ads_router_status_record_interval_timer(IN := NOT ads_router_status_record_interval_timer.Q);
fb_get_router_status_report := fb_get_router_status.bBusy;
fb_get_router_status(
	bExecute := ads_router_status_record_interval_timer.Q
);

IF fb_get_router_status_report AND NOT fb_get_router_status.bBusy THEN
	MEMCPY(ADR(router_status_record_data), ADR(fb_get_router_status.info), SIZEOF(fb_get_router_status.info));
	IF GVL.tf6420_enable THEN
		fb_ads_router_status_recorder.write(ADR(router_status_record_data));
	END_IF
END_IF

SetDynamics := GVL.planar_movers[1].MCTOPLC.SET;
ActDynamics := GVL.planar_movers[1].MCTOPLC.ACT;

record_data_set_positions.a := SetDynamics.SetPos.a;
record_data_set_positions.b := SetDynamics.SetPos.b;
record_data_set_positions.c := SetDynamics.SetPos.c;
record_data_set_positions.x := SetDynamics.SetPos.x;
record_data_set_positions.y := SetDynamics.SetPos.y;
record_data_set_positions.z := SetDynamics.SetPos.z;

IF GVL.tf6420_enable THEN
	fb_mover_dynamics_recorder.write(ADR(record_data_set_positions));
END_IF

record_data_act_positions.a := ActDynamics.ActPos.a;
record_data_act_positions.b := ActDynamics.ActPos.b;
record_data_act_positions.c := ActDynamics.ActPos.c;
record_data_act_positions.x := ActDynamics.ActPos.x;
record_data_act_positions.y := ActDynamics.ActPos.y;
record_data_act_positions.z := ActDynamics.ActPos.z;

IF GVL.tf6420_enable THEN
	fb_mover_dynamics_recorder.write(ADR(record_data_act_positions));
END_IF

END_PROGRAM

// ---- POUs/model/IoT/FB_mqtt_publish.TcPOU
FUNCTION_BLOCK FB_mqtt_publish IMPLEMENTS  ITF_CoeSdoEventHandler
VAR_INPUT
END_VAR
VAR_OUTPUT
	fb_database_aps_diag    :ST_database_aps_diag;    // 書込みデータ設定用
END_VAR
VAR
	// published message
	fbMqttClient : FB_IotMqttClient;
	fbMessageQueue : FB_IotMqttMessageQueue;
	bSetParameter : BOOL := TRUE;
	bConnect : BOOL := TRUE;
	hrErrorOccurred : HRESULT; // contains the latest occurred error
	
	fbSerializer :FB_Serializer;
	
	sTopicPub : STRING(255) := 'devices/unit230/messages/events/';
	
	// for making publish event
	publish_cycle_timer :TON;
	datetime_string: STRING(39);
	
	publish_command: BOOL;
	_error_id :UDINT;
	
	_fbDatabaseRecorder : REFERENCE TO BufferedRecord;
	
END_VAR


// Connect MQTT broker and publish

IF bSetParameter THEN
	bSetParameter := FALSE;
	fbMqttClient.sHostName := 'IndustrialOPNFair2024-IoTHub.azure-devices.net';
	fbMqttClient.nHostPort := 8883;
	fbMqttClient.stTLS.sCA := 'c:\TwinCAT\3.1\Config\Certificates\BaltimoreCyberTrust.cer'; // CA certificate 
	fbMqttClient.sClientId := 'unit230';
	fbMqttClient.stTLS.sAzureSas := 'HostName=IndustrialOPNFair2024-IoTHub.azure-devices.net;DeviceId=unit230;SharedAccessSignature=SharedAccessSignature sr=IndustrialOPNFair2024-IoTHub.azure-devices.net%2Fdevices%2Funit230&sig=aZHGqBLbPbZ0nCj3%2BrwgAJAAhzI2BvVoTXPMA%2BaobPA%3D&se=1734308970'; // Device SAS Token
	fbMqttClient.stTLS.bNoServerCertCheck:=TRUE;
	(*
	//fbMqttClient.stTLS.sCA := 'c:\TwinCAT\3.1\Config\Certificates\BaltimoreCyberTrust.crt'; // CA certificate 
	//fbMqttClient.stTLS.sAzureSas := 'HostName=IndustrialOPNFair2024-IoTHub.azure-devices.net;DeviceId=unit230;SharedAccessSignature=SharedAccessSignature sr=IndustrialOPNFair2024-IoTHub.azure-devices.net%2Fdevices%2Funit230&sig=GxT9x70t1Q1per9XXu4Az%2FJhK1jBZt14KJ%2B7LG4NB%2Fw%3D&se=1712921181'; // Device SAS Token
	fbMqttClient.sClientId := 'unit230';
	fbMqttClient.sHostName := '192.168.1.20';
	fbMqttClient.nHostPort := 1883;
	*)
	fbMqttClient.ipMessageQueue := fbMessageQueue;
END_IF

fbMqttClient.Execute(bConnect);
IF fbMqttClient.bError THEN
  // add your error logging here
  hrErrorOccurred := fbMqttClient.hrErrorCode;
END_IF


publish_cycle_timer(IN := NOT publish_command, PT := T#5S);

IF publish_cycle_timer.Q THEN
	publish_command := TRUE;
END_IF

PROPERTY fbDatabaseRecorder : REFERENCE TO BufferedRecord
SET
_fbDatabaseRecorder REF= fbDatabaseRecorder;
END_SET
END_PROPERTY

{warning 'add property implementation'}
PROPERTY nErrID : UDINT
GET
nErrID := _error_id;
END_GET
END_PROPERTY

{warning 'add method implementation '}
METHOD sdo_data_received : BOOL
VAR_INPUT
	command	: REFERENCE TO bajp_diagtool.CoeSdoCommand;
END_VAR
VAR
	diag_data_body: POINTER TO sdo_xplanar_aps_diag;
	temp: UDINT;
	i: UINT;
END_VAR
VAR_INST
	tile_number : UINT;
	sPayloadPub : STRING(255);
	pub_complete : ARRAY [1..2] OF BOOL;
	// Record data buffer
END_VAR
diag_data_body := command.pDstBuf;
CASE command.nSlaveAddr OF
	1001:
		tile_number := 1;
	1003:
		tile_number := 2;
END_CASE

//For TF6420 Database
IF __ISVALIDREF(_fbDatabaseRecorder) THEN
	fb_database_aps_diag.tile_number := TO_STRING(tile_number);
	fb_database_aps_diag.acceleration_y := diag_data_body^.acceleration_y;
	fb_database_aps_diag.acceleration_y := diag_data_body^.acceleration_y;
	fb_database_aps_diag.acceleration_z := diag_data_body^.acceleration_z;
	fb_database_aps_diag.auxiliary_voltage := diag_data_body^.auxiliary_voltage;
	fb_database_aps_diag.dc_link_voltage := diag_data_body^.dc_link_voltage;
	fb_database_aps_diag.fan_duty_cycle := diag_data_body^.fan_duty_cycle;
	fb_database_aps_diag.fan_rpm := diag_data_body^.fan_rpm;
	fb_database_aps_diag.fb_fw_rev := diag_data_body^.fb_fw_rev;
	fb_database_aps_diag.power_supply_current := diag_data_body^.power_supply_current;
	fb_database_aps_diag.supply_voltage_us := diag_data_body^.supply_voltage_us;
	fb_database_aps_diag.temperature_center := diag_data_body^.temperature_center;
	fb_database_aps_diag.temperature_east := diag_data_body^.temperature_east;
	fb_database_aps_diag.temperature_north := diag_data_body^.temperature_north;
	fb_database_aps_diag.temperature_power := diag_data_body^.temperature_power;
	fb_database_aps_diag.temperature_south := diag_data_body^.temperature_south;
	fb_database_aps_diag.temperature_west := diag_data_body^.temperature_west;
	fb_database_aps_diag.time_to_shutdown := diag_data_body^.time_to_shutdown;
	IF GVL.tf6420_enable THEN
		_fbDatabaseRecorder.write(ADR(fb_database_aps_diag));
	END_IF
END_IF


// For TF6701 MQTT
IF publish_command AND fbMqttClient.bConnected THEN
	datetime_string := SYSTEMTIME_TO_ISO8601(
		systemTime := command.datetime,
		nBias := 0,
		bUTC := TRUE,
		nPrecision := 3
	);
	CASE tile_number OF
		1:
			temp := diag_data_body^.temperature_west;
		2:
			temp := diag_data_body^.temperature_east;
	END_CASE
	sPayloadPub := fbSerializer.serialize(
	  datetime := datetime_string,
	  device_name := CONCAT('xplanar_tile_', UINT_TO_STRING(tile_number)),
	  temp := temp,
	  fan_rpm := diag_data_body^.fan_rpm,
	  current := diag_data_body^.power_supply_current
	);
	IF fbMqttClient.Publish(	sTopic:= sTopicPub, 
				pPayload:= ADR(sPayloadPub), nPayloadSize:= LEN2(ADR(sPayloadPub)), 
				eQoS:= TcIotMqttQos.AtMostOnceDelivery, bRetain:= FALSE, bQueue:= FALSE ) THEN
		_error_id := 0;
		sdo_data_received := TRUE;
	END_IF
    IF fbMqttClient.bError THEN
      // add your error logging here
    	_error_id := TO_UDINT(fbMqttClient.hrErrorCode);
	  	sdo_data_received := TRUE;
	ELSE
		pub_complete[tile_number] := TRUE;
    END_IF
	publish_command := FALSE;
	FOR i := 1 TO 2 DO
		IF NOT pub_complete[i] THEN
			publish_command := TRUE;
		END_IF
	END_FOR
ELSE
	FOR i := 1 TO 2 DO
		pub_complete[i] := FALSE;
	END_FOR
	sdo_data_received := TRUE;
END_IF
END_METHOD

END_FUNCTION_BLOCK

// ---- POUs/model/IoT/FB_serializer.TcPOU
FUNCTION_BLOCK FB_serializer
VAR_INPUT
END_VAR
VAR_OUTPUT
END_VAR
VAR
  fbJson  : FB_JsonSaxWriter;
END_VAR

METHOD serialize : STRING(255)
VAR_INPUT
  datetime: STRING;
  device_name: STRING;
  temp: UDINT;
  fan_rpm: UDINT;
  current: DINT;
END_VAR
fbJson.StartObject();       // ‘{‘ の出力
fbJson.AddKey('datetime');
fbJson.AddString(datetime);
fbJson.AddKey('device_name');
fbJson.AddString(device_name);
fbJson.AddKey('temperature');		//キー temperature: の出力
fbJson.AddUdint(temp); // 温度出力
fbJson.AddKey('fan_rpm');		//キー temperature: の出力
fbJson.AddUdint(fan_rpm); // FAN回転数出力
fbJson.AddKey('current');		//キー temperature: の出力
fbJson.AddDint(current); // 電流値
fbJson.EndObject();			// ‘}’ の出力
serialize := fbJson.GetDocument();	// 文字列へ出力
fbJson.ResetDocument();		// SAXバッファクリア
END_METHOD

END_FUNCTION_BLOCK

// ---- GlobalTextList.TcGTLO
TEXTLIST GlobalTextList
  883 = '%0.1f %'
  949 = '%0.1f deg'
  769 = '%0.1f ℃'
  777 = '%0.2f'
  534 = '%0d'
  623 = '%0f'
  142 = '%1d'
  268 = '%1d '
  622 = '%1d RPM'
  178 = '%2f'
  584 = '%s'
  462 = '0°'
  368 = '180°'
  471 = '270°'
  767 = '90°'
  759 = 'A1'
  909 = 'A2'
  847 = 'A3'
  33 = 'Auto Start'
  864 = 'B1'
  838 = 'B2'
  280 = 'B3'
  335 = 'C1'
  876 = 'C2'
  954 = 'C3'
  223 = 'Center: %'
  75 = 'Center: %0.1f deg'
  364 = 'Center: %0.2f deg'
  921 = 'Cycle duty:  %0d %'
  602 = 'Cycle duty:  %1d %'
  920 = 'Disable'
  794 = 'Duty:  %0d %'
  929 = 'Enable'
  209 = 'Enable/ Reset'
  112 = 'Error'
  535 = 'Initilalize'
  166 = 'IoT Record'
  900 = 'L1'
  522 = 'L2'
  983 = 'L3'
  589 = 'Left: %0.1f deg'
  697 = 'mA'
  869 = 'Manual mode'
  610 = 'Manual Mode'
  989 = 'Power current:  %0d mA'
  383 = 'PWM %0.1f %'
  35 = 'PWM %0d %'
  821 = 'Reset'
  384 = 'RPM'
  689 = 'Run'
  145 = 'Stop'
  311 = 'test'
  296 = 'UP'
  636 = 'イベント'
  518 = 'ジョブID'
  415 = 'ジョブ動作'
  822 = 'ジョブ履歴'
  34 = 'スタート'
  898 = 'タイル2'
  385 = 'タスク'
  657 = 'タスク名'
  237 = 'タスク種別'
  536 = 'マニュアル動作'
  481 = 'マニュアル動作パターン登録と実行'
  911 = 'マニュアル登録と実行'
  40 = 'メイン'
  257 = 'レシピ登録と実行'
  680 = 'レシピ登録画面'
  798 = '前傾'
  765 = '右タイル'
  621 = '右傾'
  391 = '左タイル'
  298 = '左傾'
  140 = '後傾'
  320 = '指令:  %1d %'
  262 = '操作'
  521 = '操作画面'
  499 = '時刻'
  523 = '水平'
  450 = '消費電流: '
  183 = '消費電流:  %0d mA'
  362 = '現在の動作 : %s'
  755 = '登録処理内容'
END_TEXTLIST

// ---- VISUs/ActionMode.TcTLO
TEXTLIST ActionMode
  1 = '直線動作(MoveToPosition)'
  2 = '回転動作(MoveC)'
  3 = '上下動作(MoveZ)'
  4 = '前後動作(MoveA)'
  5 = '左右動作(MoveB)'
  6 = '前後左右(MoveA/B混合)'
   = ''
END_TEXTLIST

// ---- VISUs/MachineMode.TcTLO
TEXTLIST MachineMode
  0 = '電源OFF'
  1 = 'ジョブ初期化'
  2 = '原点復帰ジョブ作成'
  3 = '原点復帰中'
  4 = '連続ジョブ作成'
  5 = '原点復帰完了'
  6 = 'デモモード'
  7 = 'マニュアルモード'
   = ''
END_TEXTLIST

// ---- VISUs/Visualization.TcVIS
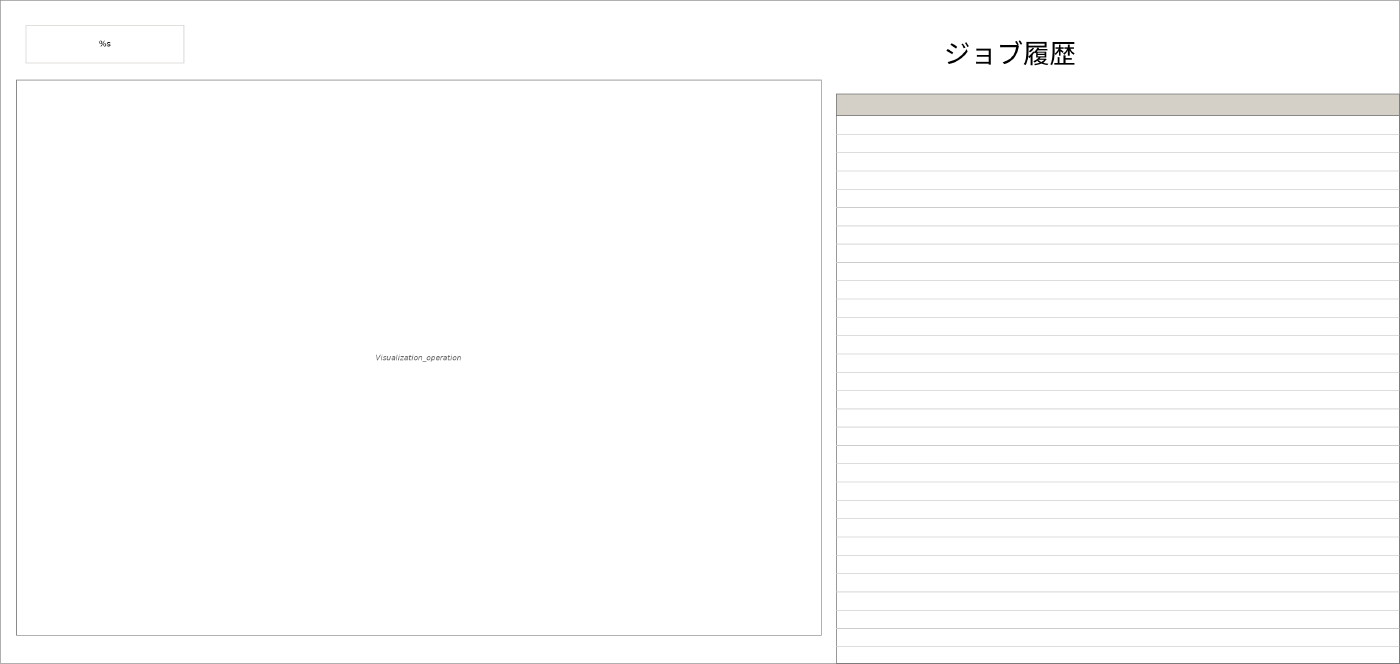
VISUALIZATION Visualization  // 1911x907
    TabControl (22,109 1099x759)
        shows Visualization_operation()
        shows Visualization_recipe()
        [0]: TabTitle=メイン
        [1]: TabTitle=マニュアル動作
    Table (1141,128 770x779), data array: MAIN.ads_reporter.log_view
        p3854506369: MAIN.ads_reporter.log_view[0,INDEX]
        p1892666644: MAIN.ads_reporter.log_view[1,INDEX]
        p2232123230: 時刻
        p511219082: タスク名
        p2685023577: MAIN.ads_reporter.log_view[INDEX]
        p338671338: MAIN.ads_reporter.log_view[3,INDEX]
        p1755163831: ジョブID
        p2170511999: MAIN.ads_reporter.log_view[2,INDEX]
        p4092479075: イベント
    Label (1164,50 429x47), "ジョブ履歴"
    Textfield (35,34 216x52), "%s", text list: 'MachineMode', text index: MAIN.machine_mode
END_VISUALIZATION

// ---- VISUs/Visualization_operation.TcVIS
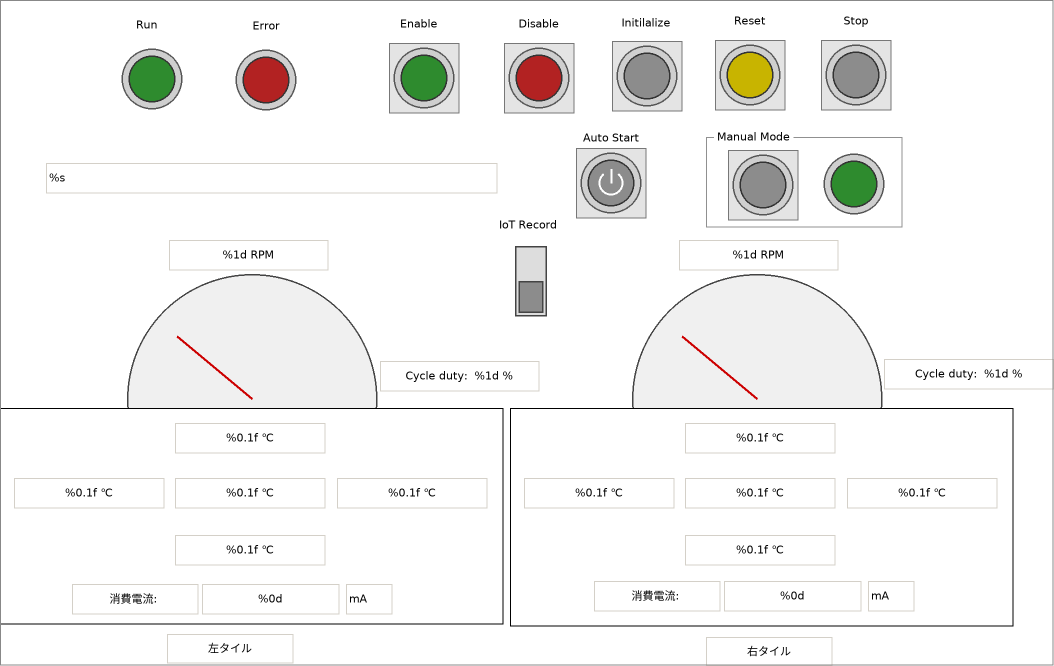
VISUALIZATION Visualization_operation  // 1054x666
    PushSwitch (389,43 70x70), variable: MAIN.bEnable, behaviour: TAP, style: Switch-PushSwitch-Green
    Label (369,9 100x30), "Enable"
    PushSwitch (504,43 70x70), variable: MAIN.bDisable, behaviour: TAP, style: Switch-PushSwitch-Red
    Label (489,9 100x30), "Disable"
    Lamp1 (117,44 70x70), variable: MAIN.ServoON, style: Lamp-Lamp1-Green
    Lamp1 (231,45 70x70), variable: MAIN.Error, style: Lamp-Lamp1-Red
    Label (97,0 100x50), "Run"
    Label (216,1 100x50), "Error"
    PushSwitch (715,40 70x70), variable: MAIN.bReset, behaviour: TOGGLE, style: Switch-PushSwitch-Yellow
    Label (700,6 100x30), "Reset"
    PushSwitch (821,40 70x70), variable: MAIN.bStop, behaviour: TAP, style: Switch-PushSwitch-Gray
    Label (806,6 100x30), "Stop"
    Meter180 (632,274 250x250), value: IoT.planar_tiles_diag_data[1].fan_rpm, style: Meter-Meter180-Gray, scale format: %1d, scale 0..3000
    Meter180 (127,274 250x250), value: IoT.planar_tiles_diag_data[2].fan_rpm, style: Meter-Meter180-Gray, scale format: %1d, scale 0..3000
    RoundedRectangle (0,408 503x216)
    Textfield (14,478 150x30), "%0.1f ℃", text variable: IoT.planar_tiles_diag_data[2].temperature_west / 10.0
    Textfield (175,478 150x30), "%0.1f ℃", text variable: IoT.planar_tiles_diag_data[2].temperature_center / 10.0
    Textfield (337,478 150x30), "%0.1f ℃", text variable: IoT.planar_tiles_diag_data[2].temperature_east / 10.0
    Textfield (175,423 150x30), "%0.1f ℃", text variable: IoT.planar_tiles_diag_data[2].temperature_north / 10.0
    Textfield (175,535 150x30), "%0.1f ℃", text variable: IoT.planar_tiles_diag_data[2].temperature_south / 10.0
    RoundedRectangle (510,408 503x218)
    Textfield (524,478 150x30), "%0.1f ℃", text variable: IoT.planar_tiles_diag_data[1].temperature_west / 10.0
    Textfield (685,478 150x30), "%0.1f ℃", text variable: IoT.planar_tiles_diag_data[1].temperature_center / 10.0
    Textfield (847,478 150x30), "%0.1f ℃", text variable: IoT.planar_tiles_diag_data[1].temperature_east / 10.0
    Textfield (685,423 150x30), "%0.1f ℃", text variable: IoT.planar_tiles_diag_data[1].temperature_north / 10.0
    Textfield (685,535 150x30), "%0.1f ℃", text variable: IoT.planar_tiles_diag_data[1].temperature_south / 10.0
    Textfield (202,584 137x30), "%0d", text variable: IoT.planar_tiles_diag_data[2].power_supply_current / 10.0
    Textfield (72,584 126x30), "消費電流:"
    Textfield (346,584 46x30), "mA"
    Textfield (724,581 137x30), "%0d", text variable: IoT.planar_tiles_diag_data[1].power_supply_current / 10.0
    Textfield (594,581 126x30), "消費電流:"
    Textfield (868,581 46x30), "mA"
    Textfield (706,637 126x29), "右タイル"
    Textfield (167,634 126x29), "左タイル"
    Textfield (380,361 159x30), "Cycle duty: %1d %", text variable: IoT.planar_tiles_diag_data[2].fan_duty_cycle
    Textfield (884,359 170x30), "Cycle duty: %1d %", text variable: IoT.planar_tiles_diag_data[2].fan_duty_cycle
    Textfield (169,240 159x30), "%1d RPM", text variable: IoT.planar_tiles_diag_data[2].fan_rpm
    Textfield (679,240 159x30), "%1d RPM", text variable: IoT.planar_tiles_diag_data[1].fan_rpm
    Textfield (46,163 451x30), "%s", text variable: MAIN.ads_reporter.executing.task_name
    PushSwitch (612,41 70x70), variable: MAIN.Init_Start, behaviour: TOGGLE, style: Switch-PushSwitch-Gray
    Label (596,8 100x30), "Initilalize"
    Label (561,123 100x30), "Auto Start"
    GroupBox (706,129 196x98), "Manual Mode"
        Lamp1 (113,20 70x70), variable: MAIN.manu_mode, style: Lamp-Lamp1-Green
        PushSwitch (22,21 70x70), variable: MAIN.manu_mode, behaviour: TOGGLE, style: Switch-PushSwitch-Gray
    Lamp1 (819,149 70x70), variable: MAIN.manu_mode, style: Lamp-Lamp1-Green
    PushSwitch (728,150 70x70), variable: MAIN.manu_mode, behaviour: TOGGLE, style: Switch-PushSwitch-Gray
    DipSwitch (496,246 70x70), variable: GVL.tf6420_enable, behaviour: TOGGLE, style: Switch-DipSwitch-Gray
    Label (478,210 100x30), "IoT Record"
    PowerSwitch (576,148 70x70), variable: MAIN.Demo_Start, behaviour: TOGGLE, style: Switch-PowerSwitch-Gray
END_VISUALIZATION

// ---- VISUs/Visualization_recipe.TcVIS
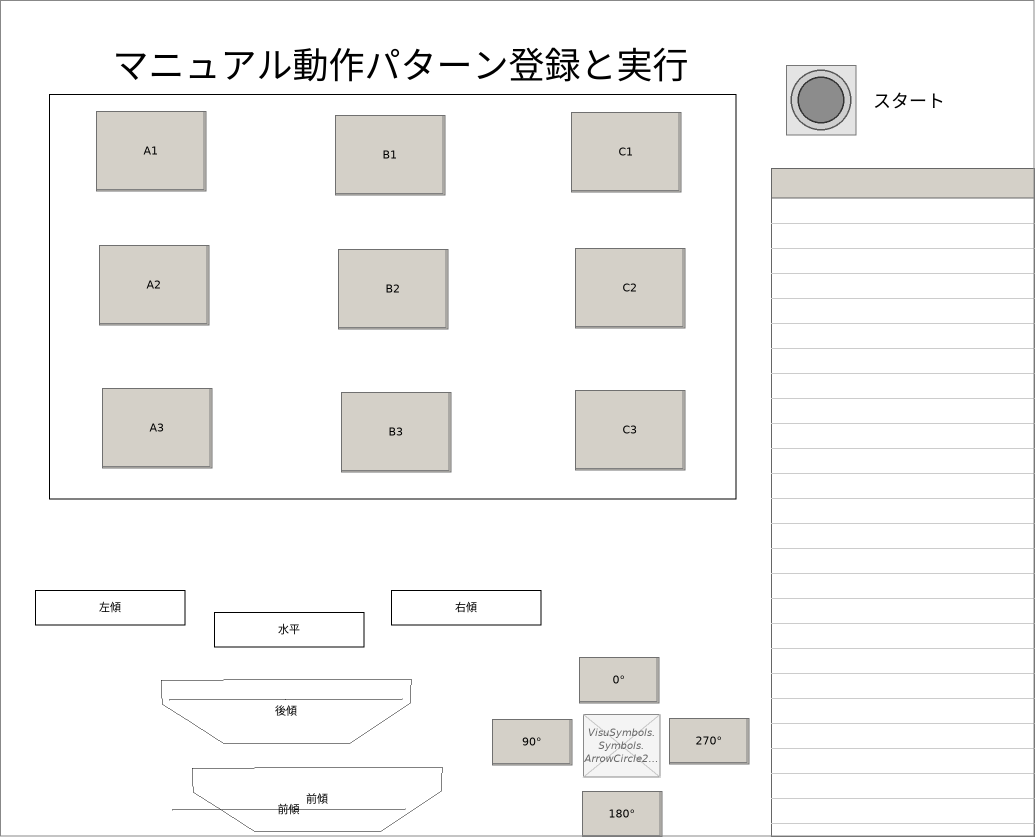
VISUALIZATION Visualization_recipe  // 1035x837
    RoundedRectangle (49,94 687x405)
    Button (575,390 110x80), "C3"
        tap MAIN.manupilator_buttons[8]
    Button (575,248 110x80), "C2"
        tap MAIN.manupilator_buttons[7]
    Button (571,112 110x80), "C1"
        tap MAIN.manupilator_buttons[6]
    Button (335,115 110x80), "B1"
        tap MAIN.manupilator_buttons[5]
    Button (338,249 110x80), "B2"
        tap MAIN.manupilator_buttons[4] p3779583253=TRUE
    Button (341,392 110x80), "B3"
        tap MAIN.manupilator_buttons[3]
    Button (96,111 110x80), "A1"
        tap MAIN.manupilator_buttons[2]
    Button (99,245 110x80), "A2"
        tap MAIN.manupilator_buttons[1]
    Button (102,388 110x80), "A3"
        tap MAIN.manupilator_buttons[0]
    Polyline (44,593) (45,594)
    RoundedRectangle (35,590 150x35), angle 330, "左傾"
        tap MAIN.manupilator_buttons[14] p3779583253=TRUE
    RoundedRectangle (391,590 150x35), angle 30, "右傾"
        tap MAIN.manupilator_buttons[13]
    Polygon (161,680) (411,679) (410,703) (350,743) (223,743) (189,721) (162,704), "後傾"
        tap MAIN.manupilator_buttons[12]
    Polyline (402,699) (169,700)
    Polygon (192,768) (442,767) (441,791) (381,831) (254,831) (220,809) (193,792), "前傾"
        tap MAIN.manupilator_buttons[11] p3779583253=TRUE
    Polyline (405,809) (172,810), "前傾"
    Table (771,168 264x669), data array: MAIN.Recipe_Display
        p1128707560: jobmgmt.ParamFuturesLib.MAX_TASK_NUM
        p3854506369: MAIN.Recipe_Display[INDEX]
        p2232123230: 登録処理内容
    Label (94,42 613x47), "マニュアル動作パターン登録と実行"
    PushSwitch (786,65 70x70), variable: MAIN.manual_start, behaviour: TAP, style: Switch-PushSwitch-Gray
    Label (868,78 82x47), "スタート"
    RoundedRectangle (214,612 150x35), "水平"
        tap MAIN.manupilator_buttons[15]
    Image (583,714 77x63), image: VisuSymbols.Symbols.ArrowCircle2LeftRightLeft
    Button (492,719 80x46), "90°"
        tap MAIN.manupilator_buttons[16]
    Button (579,657 80x46), "0°"
        tap MAIN.manupilator_buttons[17]
    Button (669,718 80x46), "270°"
        tap MAIN.manupilator_buttons[18]
    Button (582,791 80x46), "180°"
        tap MAIN.manupilator_buttons[19]
END_VISUALIZATION
